KUKA KRL program: STOP_SONG.src, STOP_SONG.dat

--- STOP_SONG.src ---
&ACCESS RVO
&REL 18
&PARAM DISKPATH = KRC:\R1\Program\_KLAVIRISTA_V2\subprogram
DEF  STOP_SONG ( )
;FOLD INI
   IF NOT $ON_PATH THEN
  ;FOLD BASISTECH INI
    GLOBAL INTERRUPT DECL 3 WHEN $STOPMESS==TRUE DO IR_STOPM ( )
    INTERRUPT ON 3
    BAS (#INITMOV,0 )
  ;ENDFOLD (BASISTECH INI)
  ENDIF
;ENDFOLD (INI)
BRAKE
$OUT[8]=TRUE
IF $TIMER_STOP[5] THEN
WAIT SEC 2
WAIT FOR ( $IN[7] OR PyACK)
ELSE
PyWAIT = TRUE
$TIMER_STOP[5]=TRUE
$TIMER[6]=0
$TIMER_STOP[6]=FALSE
REPEAT
   WAIT SEC 5 ; 2*BAR=5000 = 5s
UNTIL ( $IN[7] OR PyACK)
$TIMER_STOP[5]=FALSE
$TIMER_STOP[6]=TRUE
PyWAIT=FALSE
ENDIF
PULSE($OUT[7], TRUE, 0.5) ;reset ACK
PyACK=FALSE
WAIT FOR NOT $IN[8]
$OUT[8]=FALSE
END

--- STOP_SONG.dat ---
&ACCESS RVO
&REL 18
&PARAM DISKPATH = KRC:\R1\Program\_KLAVIRISTA_V2\subprogram
DEFDAT  STOP_SONG
;FOLD EXTERNAL DECLARATIONS;%{PE}%MKUKATPBASIS,%CEXT,%VCOMMON,%P
;FOLD BASISTECH EXT;%{PE}%MKUKATPBASIS,%CEXT,%VEXT,%P
EXT  BAS (BAS_COMMAND  :IN,REAL  :IN )
DECL INT NEXTBAR
;ENDFOLD (BASISTECH EXT)
;FOLD USER EXT;%{E}%MKUKATPUSER,%CEXT,%VEXT,%P
;Make your modifications here

;ENDFOLD (USER EXT)
;ENDFOLD (EXTERNAL DECLARATIONS)

DECL MODULEPARAM_T LAST_TP_PARAMS = {PARAMS[] "Kuka.VelocityFieldEnabled=True; Kuka.ColDetectFieldEnabled=True; Kuka.MovementParameterFieldEnabled=True; Kuka.IsAngleEnabled=False; Kuka.VelocityPtp=17; Kuka.BlendingEnabled=False; Kuka.APXEnabled=False; Kuka.CurrentCDSetIndex=0; Kuka.PointName=P66; Kuka.FrameData.base_no=0; Kuka.FrameData.tool_no=1; Kuka.FrameData.ipo_frame=#BASE; Kuka.isglobalpoint=False; Kuka.MoveDataPtpName=PDAT54; Kuka.MovementDataPdat.apo_mode=#CDIS; Kuka.MovementDataPdat.apo_dist=500; Kuka.MovementData.vel=1; Kuka.MovementData.acc=100; Kuka.MovementData.exax_ign=0; Kuka.FrameData.point2=; Kuka.MoveDataName=CPDAT15; Kuka.MovementData.apo_fac=50; Kuka.MovementData.apo_dist=500; Kuka.MovementData.axis_acc=100; Kuka.MovementData.axis_vel=100; Kuka.MovementData.circ_typ=#BASE; Kuka.MovementData.jerk_fac=50; Kuka.MovementData.ori_typ=#VAR; Kuka.VelocityPath=1; Kuka.MovementData.cb={AUX_PT {ORI #CONSIDER,E1 #CONSIDER,E2 #CONSIDER,E3 #CONSIDER,E4 #CONSIDER,E5 #CONSIDER,E6 #CONSIDER},TARGET_PT {ORI #INTERPOLATE,E1 #INTERPOLATE,E2 #INTERPOLATE,E3 #INTERPOLATE,E4 #INTERPOLATE,E5 #INTERPOLATE,E6 #INTERPOLATE}}; Kuka.HelpPointName=P17; Kuka.Logics.Io=1; Kuka.Logics.IoName=; Kuka.Logics.State=True; Kuka.Logics.Cont=False; Kuka.Logics.Time=0.5                                                                                                                                                                                                          "}
ENDDAT
